PROGRAM extMarksPrg
VAR
    fbLogMark	: FB_RTMon_LogMarkBase;	
	
	// user defined context
	idModule1 : UINT := 10001;	

		
	// Marks
	markCounter  : ST_RTMon_MarkDef := (nContextId := idModule1, nGroupId := 1, nEventId := 0); 
END_VAR

//fbLogMark.LogMarkEx(markCounter, TcMarkOption.Start OR TcMarkOption.RefToCaller);
IF GVL.fbCrititcalSection.Enter() THEN
	GVL.iGlobalCounter:=GVL.iGlobalCounter+1;
	ConsumeTime(50);
    GVL.fbCrititcalSection.Leave();
END_IF
//fbLogMark.LogMarkEx(markCounter, TcMarkOption.Stop OR TcMarkOption.RefToCaller);

END_PROGRAM

(* stored: Version 1.1.0.1, ProductVersion 3.1.4024.11
   POU extMarksPrg: Id {254fce39-b20e-4600-bfbd-cf8c6f7bc85a}, SpecialFunc None *)
